FUNCTION_BLOCK FB_LinkDataReal EXTENDS FB_LinkDevice
VAR	
	ControlData			AT %Q* : REAL; //{simulation-interface}	
	StatusData			AT %I* : REAL; //{simulation-interface}	
END_VAR

SUPER^();

METHOD INTERNAL SetLinkStatusData : BOOL
VAR_INPUT
	fStatusData : REAL;
END_VAR
StatusData := fStatusData;
END_METHOD

METHOD INTERNAL GetLinkControlData : REAL
GetLinkControlData := ControlData;
END_METHOD

END_FUNCTION_BLOCK

(* stored: Version 1.1.0.1, ProductVersion 3.1.4024.12
   POU FB_LinkDataReal: Id {f50d67ec-1ac9-0534-2c34-45357d634bf8}, SpecialFunc None
   Method SetLinkStatusData: Id {55afac42-795a-06a9-1d86-4d027637fbd8}
   Method GetLinkControlData: Id {a6bb0f73-7f3a-0718-2ab4-b887f70d17f7} *)
